(* CoDeSys 2.3 export: STFB_MODBUSMASTER.EXP *)

(* Data type *)
TYPE stFB_ModbusMaster :
STRUCT
	byCurrentModbusSlaveAdress: BYTE;
	bModbusAddressExist: BOOL;
	bModbusCommunicationActive: BOOL;
	stCurrentDeviceSpace:  ARRAY [0..uiMaxCurrentDeviceSpace] OF stDeviceSpace;
	iNumberOfData: INT;
	bError: BOOL;
	eError: INT;
END_STRUCT
END_TYPE
